Fanuc KAREL source: ka00109.KL

-- PROVISIONAL review KL for V1013-1; original PC SHA256 61c6549e94e07de25fe95c80d89f9cdb3cd63319ba53687f3e3c6c07cbb94e3d
-- Incomplete behavior may be omitted. Consult companion uncertainty JSON. Do not deploy.
PROGRAM KA00109
%NOLOCKGROUP
VAR
  DST : INTEGER
-- UNRESOLVED_DECL SRC type=00001c
BEGIN
  -- UNRESOLVED_PC offsets 5-15; opcodes 9D,22,A5
  -- UNRESOLVED_PC offsets 20-32; opcodes 21,23
  -- UNRESOLVED_PC offsets 37-41; opcodes 7F
END KA00109
